FUNCTION_BLOCK FB_909
VAR_IN_OUT

	IG : ST_VG;

END_VAR
VAR_INPUT

	PG : ST_VG;

END_VAR
VAR_OUTPUT
END_VAR
VAR
	rMaxPressure: REAL := 5E-2;
	rMinPressure: REAL := 3E-10;

	V: REAL;
	fbGaugeState : FB_PressureState;
END_VAR

(* This function block is used to provide protection and automatic turn on of ion gauges,
 it also manages the turn on of the AT_VAC boolean, and checks to make sure the pressure is good *)

(* Real-value calculation *)
(* Generic expression for pressure in the MKS systems

P = 10^(V/0.6 -12)

*)

V := 10*INT_TO_REAL(IG.iPRESS_R)/32767;

IG.rPRESS := LREAL_TO_REAL(EXPT(10,(V-10)));


(* Protection Functions *)
(* If the PG pressure is greater than the IG.PRO_SP then the gauge is disabled *)
(* If the PG pressure is less than the IG.PRO_SP then the gauge is enabled *)
(* This FB also implements some hysteresis so the gauge doesn't have rapid power cycling while near the turn on boundary *)

IF PG.rPRESS < IG.rPRO_SP AND PG.xPRESS_OK THEN

	IG.xHV_DIS := IG.xHV_SW;

ELSIF IG.xHV_DIS THEN
	IF IG.rPRESS > IG.rPRO_SP + IG.rHYS_PR OR PG.rPRESS > IG.rPRO_SP + IG.rHYS_PR THEN
		IG.xHV_DIS := FALSE;
		IG.xHV_SW := FALSE;
	END_IF
ELSE
	IG.xHV_DIS := FALSE;
	IG.xHV_SW := FALSE;
END_IF

(* Pressure OK check *)
fbGaugeState.i_rV := V;
fbGaugeState.i_MaxPressure := rMaxPressure;
fbGaugeState.i_MinPressure := rMinPressure;
fbGaugeState(iq_stVG:=IG);

//Backwards compatibility
IG.xPRESS_OK := (IG.eState = gc_GaugeValidState) OR IG.xBAKEOUT;

(* Setpoint evaluation *)
IG.xAT_VAC := (IG.xPRESS_OK AND (IG.rPRESS<IG.rVAC_SP)) OR IG.xBAKEOUT;

END_FUNCTION_BLOCK

(* stored: Version 1.1.0.1, ProductVersion 3.1.4020.6
   POU FB_909: Id {6704ae1a-1a21-4980-b06c-d89623cfcf41}, SpecialFunc None *)
